// TIA Portal V20 export
// export: Created 2025-09-12T17:58:00.0000000Z, ExportSetting WithDefaults
FUNCTION_BLOCK "FB200_EM_Cooling"   // FB, SCL
TITLE = EM-200: Cooling Control
AUTHOR : Dallas Levine
VERSION : 0.1
// This block contains all logic for the Cooling Equipment Module (EM-200).
// stored: AutoNumber true, IsRetain false
   VAR_INPUT
      Enable : Bool;   // Enables the block's execution.
      Valve_Demand_In : Real;   // Demand signal from the main PID controller (0.0 - 100.0 %).
   END_VAR
   VAR
      UDT : "UDT200_EM_Cooling";   // The data interface for the Cooling Equipment Module.
      Feedback_Fault_Timer : TON_TIME;   // Timer for the feedback fault delay.
   END_VAR
   VAR CONSTANT
      FEEDBACK_TOLERANCE : Real := 10.0;   // Allowable deviation between command and feedback (%).
      FEEDBACK_DELAY : Time := T#60s;   // Time delay before a feedback mismatch becomes an alarm.
   END_VAR
BEGIN
   REGION Main Logic 
   IF #Enable THEN

    (/**/) #UDT.CHW_Valve_Cmd_AO := #Valve_Demand_In;

    (/**/) #UDT.CHW_Freeze_Alm := #UDT.CHW_Freeze_Stat_DI;
    IF #UDT.CHW_Freeze_Alm THEN
     #UDT.CHW_Valve_Cmd_AO := 0.0;
    END_IF;

    (/**/) #Feedback_Fault_Timer(IN:= ABS(FV:=#UDT.CHW_Valve_Cmd_AO - #UDT.CHW_Valve_Fdbk_AI) > #FEEDBACK_TOLERANCE,
           PT:= #FEEDBACK_DELAY);
    #UDT.Valve_Failure_Alm := #Feedback_Fault_Timer.Q;
   ELSE
    (/**/) #UDT.CHW_Valve_Cmd_AO := 0.0;
    #UDT.Valve_Failure_Alm := FALSE;
   END_IF;
   END_REGION
END_FUNCTION_BLOCK
